# EPICS StreamDevice protocol: celerotonChopper/celerotonChopper.proto
# Communication protocol file for Celeroton Chopper
# Mateusz Hoppe
# 2019

# choose one of the following:
Terminator = ;       # to use with real device
#Terminator = CR LF;  # to use with builded simulator

ReplyTimeout = 10;
WriteTimeout = 10;
ReadTimeout  = 10;

# ===============================================================================================================
# CONTROL SIGNALS (START/STOP/STATUS/ERROR SUPPORT)
# ===============================================================================================================

start 	  { out 0x02 0x02 0xFC; in 0x02 0x02 0xFC; }
stop 	  { out 0x02 0x03 0xFB; in 0x02 0x03 0xFB; }
getStatus {	out 0x02 0x00 0xFE;	in  0x12 0x00 "%(\$1:ERROR_CODE_1)#4r%(\$1:ERROR_CODE_2)#4r%(\$1:WARNING_CODE)#4r%(\$1:INFO_CODE)#4r%<negsum>"; }
ackErrors {	out 0x0A 0x01 "%(\$1:ERROR_CODE_1)#.4r%(\$1:ERROR_CODE_2)#.4r%<negsum>"; in  0x02 0x01 0xFD; }
sendZeros {	out 0x00 0x00 0x00 0x00 0x00 0x00 0x00 0x00 0x00 0x00 0x00 0x00 0x00 0x00 0x00 0x00; }

@replytimeout { sendZeros; }
@readtimeout  { sendZeros; }
@writetimeout { sendZeros; }
@mismatch     { sendZeros; }

# ===============================================================================================================
# READ/WRITE VARIABLES
# ===============================================================================================================

getReferenceSpeed         {	out 0x03 0x04 0x00 "%<negsum>";           in 0x07 0x04 0x03 "%#4r%<negsum>"; }
setReferenceSpeed         {	out 0x08 0x05 0x00 0x03 "%#.4r%<negsum>"; in 0x02 0x05 0xF9; }

getPhaseInductance        { out 0x03 0x04 0x0F "%<negsum>";           in 0x07 0x04 0x05 "%#4R%<negsum>"; }
setPhaseInductance        { out 0x08 0x05 0x0F 0x05 "%#.4R%<negsum>"; in 0x02 0x05 0xF9; }

getPolePairs              { out 0x03 0x04 0x09 "%<negsum>";           in 0x07 0x04 0x02 "%#4r%<negsum>"; }
setPolePairs              { out 0x08 0x05 0x09 0x02 "%#.4r%<negsum>"; in 0x02 0x05 0xF9; }

getMaxPhaseCurrent        { out 0x03 0x04 0x0A "%<negsum>";           in 0x07 0x04 0x01 "%#4r%<negsum>"; }
setMaxPhaseCurrent        { out 0x08 0x05 0x0A 0x01 "%#.4r%<negsum>"; in 0x02 0x05 0xF9; }

getMaxRotationalSpeed     {	out 0x03 0x04 0x0B "%<negsum>";           in 0x07 0x04 0x03 "%#4r%<negsum>"; }
setMaxRotationalSpeed     {	out 0x08 0x05 0x0B 0x03 "%#.4r%<negsum>"; in 0x02 0x05 0xF9; }

getSynchronizationCurrent {	out 0x03 0x04 0x0C "%<negsum>";	          in 0x07 0x04 0x02 "%#4r%<negsum>"; }
setSynchronizationCurrent {	out 0x08 0x05 0x0C 0x02 "%#.4r%<negsum>"; in 0x02 0x05 0xF9; }

getAxialMomentOfInertia   { out 0x03 0x04 0x0D "%<negsum>";           in 0x07 0x04 0x05 "%#.4R%<negsum>"; }
setAxialMomentOfInertia   { out 0x08 0x05 0x0D 0x05 "%#.4R%<negsum>"; in 0x02 0x05 0xF9; }

getPMFluxLinkage          { out 0x03 0x04 0x0E "%<negsum>";           in 0x07 0x04 0x05 "%#.4R%<negsum>"; }
setPMFluxLinkage          { out 0x08 0x05 0x0E 0x05 "%#.4R%<negsum>"; in 0x02 0x05 0xF9; }

getPhaseResistance        { out 0x03 0x04 0x10 "%<negsum>";           in 0x07 0x04 0x05 "%#.4R%<negsum>"; }
setPhaseResistance        { out 0x08 0x05 0x10 0x05 "%#.4R%<negsum>"; in 0x02 0x05 0xF9; }

getRotationDirection      { out 0x03 0x04 0x11 "%<negsum>";           in 0x07 0x04 0x02 "%#4r%<negsum>"; }
setRotationDirection      { out 0x08 0x05 0x11 0x02 "%#.4r%<negsum>"; in 0x02 0x05 0xF9; }

getAccRationAboveSync     {	out 0x03 0x04 0x12 "%<negsum>";           in 0x07 0x04 0x05 "%#.4R%<negsum>"; }
setAccRationAboveSync     {	out 0x08 0x05 0x12 0x05 "%#.4R%<negsum>"; in 0x02 0x05 0xF9; }

getAccRationBelowSync     {	out 0x03 0x04 0x13 "%<negsum>";           in 0x07 0x04 0x05 "%#.4R%<negsum>"; }
setAccRationBelowSync     {	out 0x08 0x05 0x13 0x05 "%#.4R%<negsum>"; in 0x02 0x05 0xF9; }

getSCRaiseTime            { out 0x03 0x04 0x14 "%<negsum>";           in 0x07 0x04 0x05 "%#.4R%<negsum>"; }
setSCRaiseTime            { out 0x08 0x05 0x14 0x05 "%#.4R%<negsum>"; in 0x02 0x05 0xF9; }

getUserDefSyncSpeed       { out 0x03 0x04 0x15 "%<negsum>";           in 0x07 0x04 0x02 "%#4r%<negsum>"; }
setUserDefSyncSpeed       { out 0x08 0x05 0x15 0x02 "%#.4r%<negsum>"; in 0x02 0x05 0xF9; }

getUserDefSyncSpeedL      { out 0x03 0x04 0x18 "%<negsum>";           in 0x07 0x04 0x03 "%#4r%<negsum>"; }
setUserDefSyncSpeedL      { out 0x08 0x05 0x18 0x03 "%#.4r%<negsum>"; in 0x02 0x05 0xF9; }

getUserDefSyncSpeedU      { out 0x03 0x04 0x19 "%<negsum>";           in 0x07 0x04 0x03 "%#4r%<negsum>"; }
setUserDefSyncSpeedU      { out 0x08 0x05 0x19 0x03 "%#.4r%<negsum>"; in 0x02 0x05 0xF9; }

getProportionalSpeedGain  { out 0x03 0x04 0x1B "%<negsum>";           in 0x07 0x04 0x05 "%#.4R%<negsum>"; }
setProportionalSpeedGain  { out 0x08 0x05 0x1B 0x05 "%#.4R%<negsum>"; in 0x02 0x05 0xF9; }

getIntegralSpeedGain      { out 0x03 0x04 0x1C "%<negsum>";           in 0x07 0x04 0x05 "%#.4R%<negsum>"; }
setIntegralSpeedGain      { out 0x08 0x05 0x1C 0x05 "%#.4R%<negsum>"; in 0x02 0x05 0xF9; }

getLevitate               { out 0x03 0x04 0x1D "%<negsum>";           in 0x07 0x04 0x02 "%#4r%<negsum>"; }
setLevitate               { out 0x08 0x05 0x1D 0x02 "%#.4r%<negsum>"; in 0x02 0x05 0xF9; }

# ===============================================================================================================
# READ ONLY VARIABLES
# ===============================================================================================================

getActualSpeed   	{ out 0x03 0x04 0x01 "%<negsum>"; in 0x07 0x04 0x03 "%#4r%<negsum>"; }
getDefSyncSpeedL 	{ out 0x03 0x04 0x16 "%<negsum>"; in 0x07 0x04 0x03 "%#4r%<negsum>"; }
getDefSyncSpeedU 	{ out 0x03 0x04 0x17 "%<negsum>"; in 0x07 0x04 0x03 "%#4r%<negsum>"; }
getDCLinkVoltage 	{ out 0x03 0x04 0x05 "%<negsum>"; in 0x07 0x04 0x01 "%#4r%<negsum>"; }
getDCLinkCurrent 	{ out 0x03 0x04 0x02 "%<negsum>"; in 0x07 0x04 0x01 "%#4r%<negsum>"; }
getCurrentReference { out 0x03 0x04 0x03 "%<negsum>"; in 0x07 0x04 0x01 "%#4r%<negsum>"; }
getOutputPower 		{ out 0x03 0x04 0x06 "%<negsum>"; in 0x07 0x04 0x01 "%#4r%<negsum>"; }
getConverterTemp 	{ out 0x03 0x04 0x04 "%<negsum>"; in 0x07 0x04 0x01 "%#4r%<negsum>"; }
getMotorTempTHC 	{ out 0x03 0x04 0x07 "%<negsum>"; in 0x07 0x04 0x01 "%#4r%<negsum>"; }
getMotorTempPTC 	{ out 0x03 0x04 0x08 "%<negsum>"; in 0x07 0x04 0x01 "%#4r%<negsum>"; }
